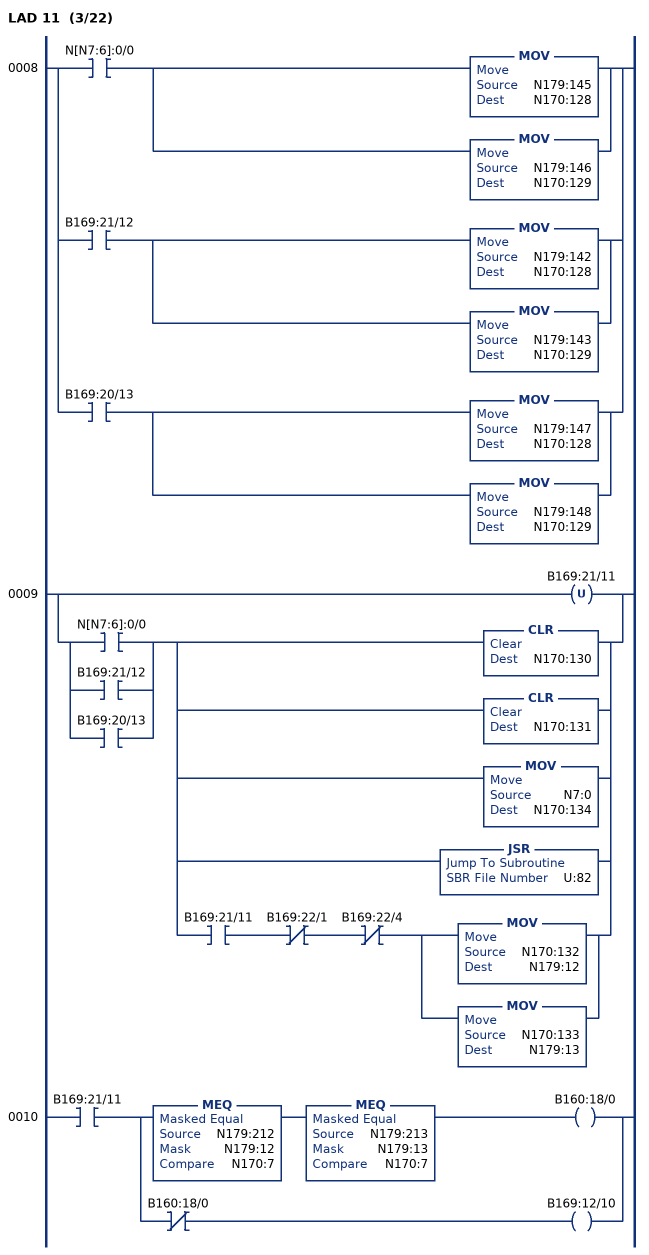
% Rung: 8 %
SOR BST XIC N[N7:6]:0/0 BST MOV N179:145 N170:128 NXB MOV N179:146 N170:129 BND NXB XIC B169:21/12 BST MOV N179:142 N170:128 NXB MOV N179:143 N170:129 BND NXB XIC B169:20/13 BST MOV N179:147 N170:128 NXB MOV N179:148 N170:129 BND BND EOR
% Rung: 9 %
SOR BST OTU B169:21/11 NXB BST XIC N[N7:6]:0/0 NXB XIC B169:21/12 NXB XIC B169:20/13 BND BST CLR N170:130 NXB CLR N170:131 NXB MOV N7:0 N170:134 NXB JSR U:82 NXB XIC B169:21/11 XIO B169:22/1 XIO B169:22/4 BST MOV N170:132 N179:12 NXB MOV N170:133 N179:13 BND BND BND EOR
% Rung: 10 %
SOR XIC B169:21/11 BST MEQ N179:212 N179:12 N170:7 MEQ N179:213 N179:13 N170:7 OTE B160:18/0 NXB XIO B160:18/0 OTE B169:12/10 BND EOR

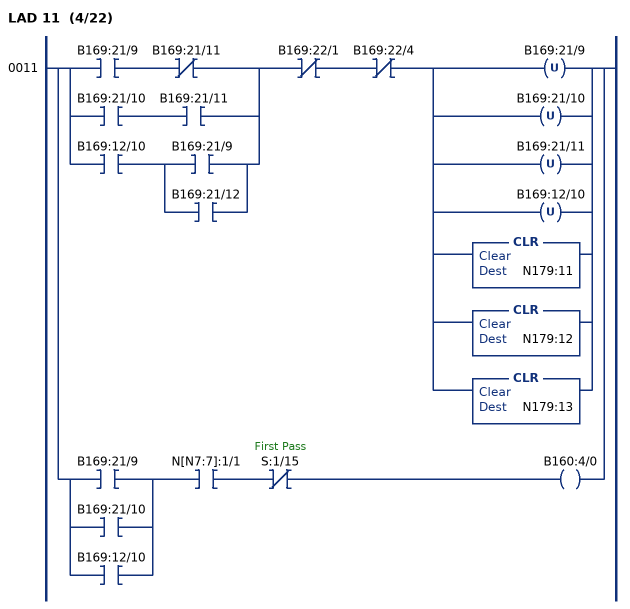
% Rung: 11 %
SOR BST BST XIC B169:21/9 XIO B169:21/11 NXB XIC B169:21/10 XIC B169:21/11 NXB XIC B169:12/10 BST XIC B169:21/9 NXB XIC B169:21/12 BND BND XIO B169:22/1 XIO B169:22/4 BST OTU B169:21/9 NXB OTU B169:21/10 NXB OTU B169:21/11 NXB OTU B169:12/10 NXB CLR N179:11 NXB CLR N179:12 NXB CLR N179:13 BND NXB BST XIC B169:21/9 NXB XIC B169:21/10 NXB XIC B169:12/10 BND XIC N[N7:7]:1/1 XIO S:1/15 OTE B160:4/0 BND EOR
%   S:1/15  "First Pass" %

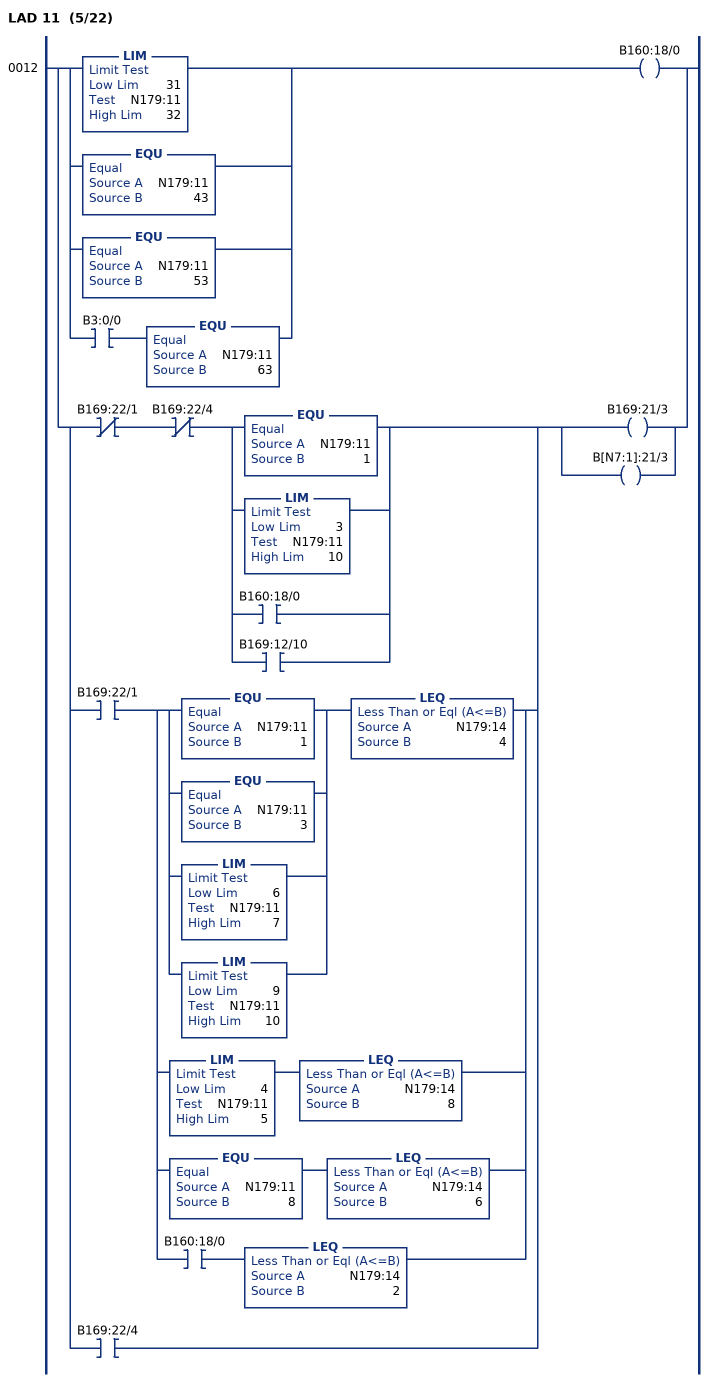
% Rung: 12 %
SOR BST BST LIM 31 N179:11 32 NXB EQU N179:11 43 NXB EQU N179:11 53 NXB XIC B3:0/0 EQU N179:11 63 BND OTE B160:18/0 NXB BST XIO B169:22/1 XIO B169:22/4 BST EQU N179:11 1 NXB LIM 3 N179:11 10 NXB XIC B160:18/0 NXB XIC B169:12/10 BND NXB XIC B169:22/1 BST BST EQU N179:11 1 NXB EQU N179:11 3 NXB LIM 6 N179:11 7 NXB LIM 9 N179:11 10 BND LEQ N179:14 4 NXB LIM 4 N179:11 5 LEQ N179:14 8 NXB EQU N179:11 8 LEQ N179:14 6 NXB XIC B160:18/0 LEQ N179:14 2 BND NXB XIC B169:22/4 BND BST OTE B169:21/3 NXB OTE B[N7:1]:21/3 BND BND EOR

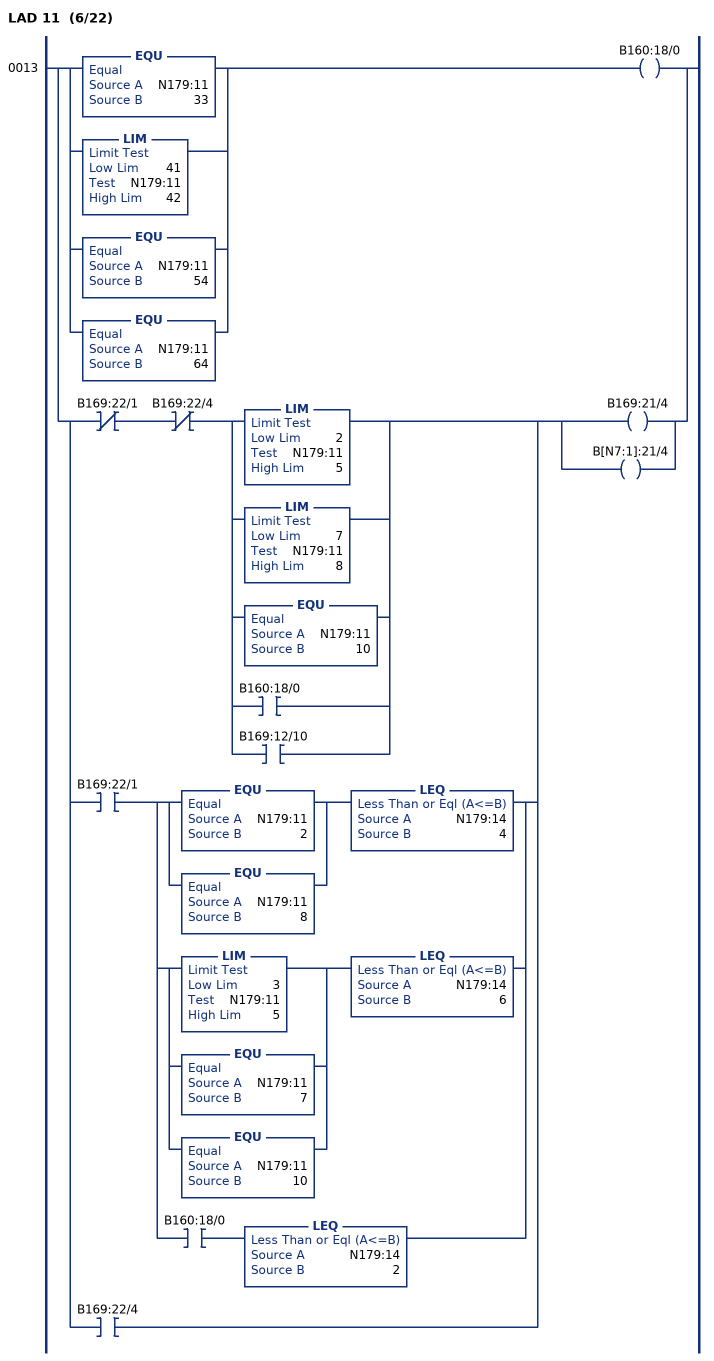
% Rung: 13 %
SOR BST BST EQU N179:11 33 NXB LIM 41 N179:11 42 NXB EQU N179:11 54 NXB EQU N179:11 64 BND OTE B160:18/0 NXB BST XIO B169:22/1 XIO B169:22/4 BST LIM 2 N179:11 5 NXB LIM 7 N179:11 8 NXB EQU N179:11 10 NXB XIC B160:18/0 NXB XIC B169:12/10 BND NXB XIC B169:22/1 BST BST EQU N179:11 2 NXB EQU N179:11 8 BND LEQ N179:14 4 NXB BST LIM 3 N179:11 5 NXB EQU N179:11 7 NXB EQU N179:11 10 BND LEQ N179:14 6 NXB XIC B160:18/0 LEQ N179:14 2 BND NXB XIC B169:22/4 BND BST OTE B169:21/4 NXB OTE B[N7:1]:21/4 BND BND EOR

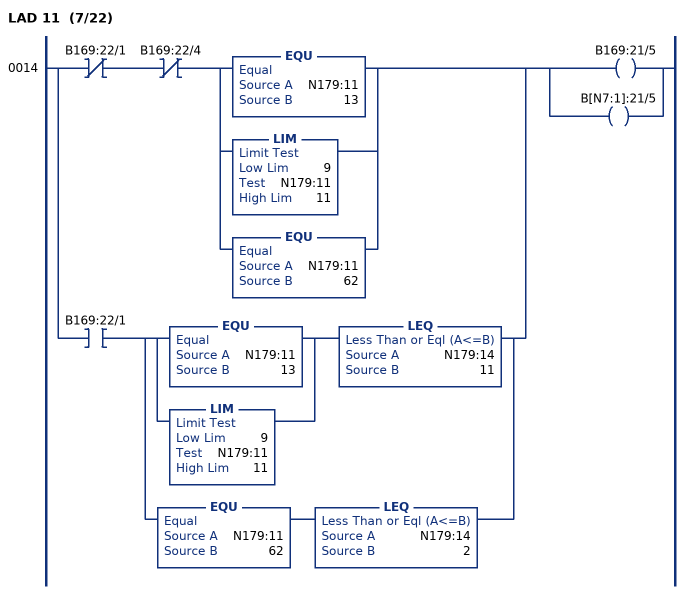
% Rung: 14 %
SOR BST XIO B169:22/1 XIO B169:22/4 BST EQU N179:11 13 NXB LIM 9 N179:11 11 NXB EQU N179:11 62 BND NXB XIC B169:22/1 BST BST EQU N179:11 13 NXB LIM 9 N179:11 11 BND LEQ N179:14 11 NXB EQU N179:11 62 LEQ N179:14 2 BND BND BST OTE B169:21/5 NXB OTE B[N7:1]:21/5 BND EOR

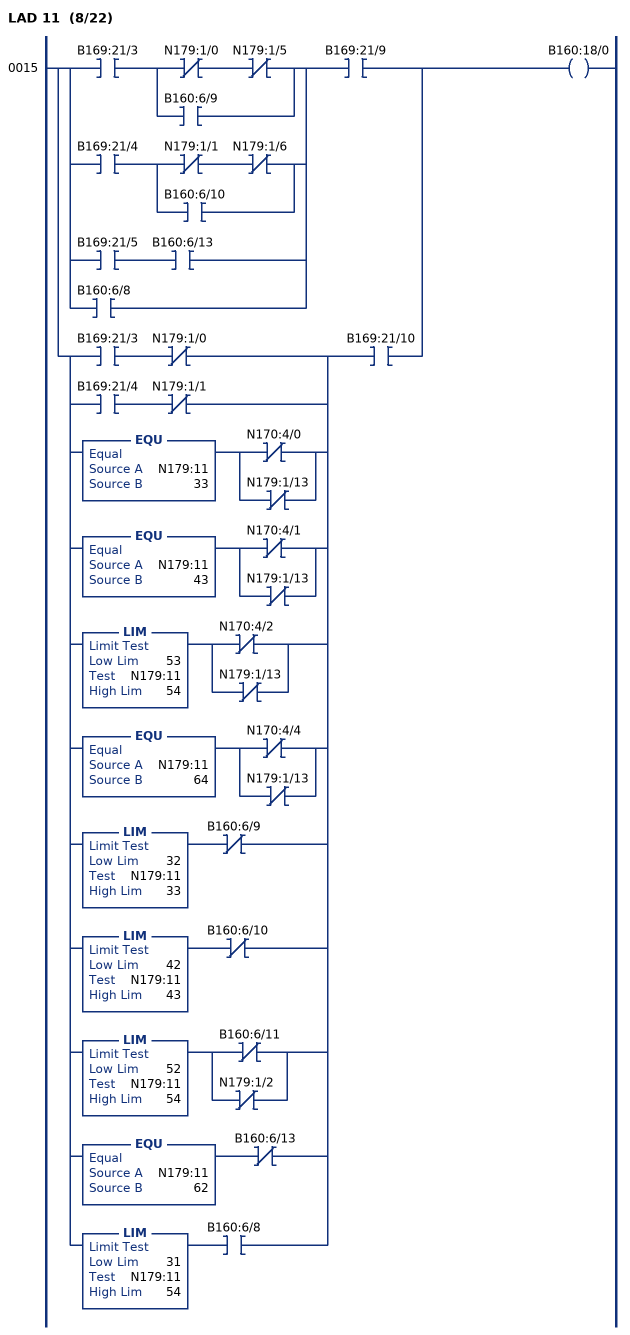
% Rung: 15 %
SOR BST BST XIC B169:21/3 BST XIO N179:1/0 XIO N179:1/5 NXB XIC B160:6/9 BND NXB XIC B169:21/4 BST XIO N179:1/1 XIO N179:1/6 NXB XIC B160:6/10 BND NXB XIC B169:21/5 XIC B160:6/13 NXB XIC B160:6/8 BND XIC B169:21/9 NXB BST XIC B169:21/3 XIO N179:1/0 NXB XIC B169:21/4 XIO N179:1/1 NXB EQU N179:11 33 BST XIO N170:4/0 NXB XIO N179:1/13 BND NXB EQU N179:11 43 BST XIO N170:4/1 NXB XIO N179:1/13 BND NXB LIM 53 N179:11 54 BST XIO N170:4/2 NXB XIO N179:1/13 BND NXB EQU N179:11 64 BST XIO N170:4/4 NXB XIO N179:1/13 BND NXB LIM 32 N179:11 33 XIO B160:6/9 NXB LIM 42 N179:11 43 XIO B160:6/10 NXB LIM 52 N179:11 54 BST XIO B160:6/11 NXB XIO N179:1/2 BND NXB EQU N179:11 62 XIO B160:6/13 NXB LIM 31 N179:11 54 XIC B160:6/8 BND XIC B169:21/10 BND OTE B160:18/0 EOR

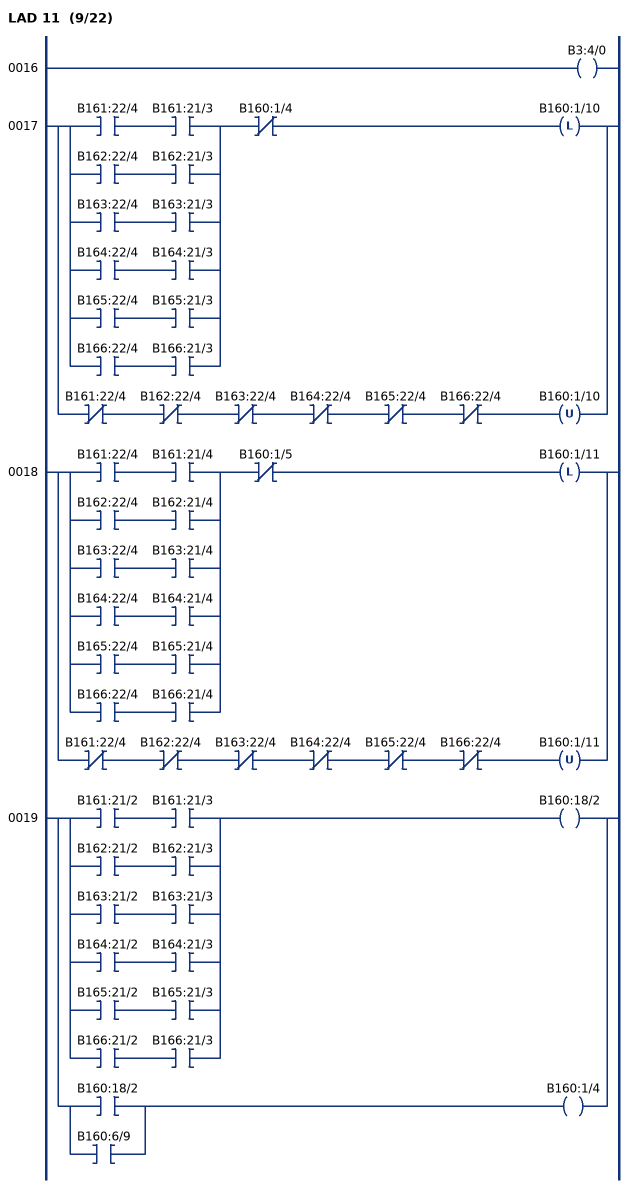
% Rung: 16 %
SOR OTE B3:4/0 EOR
% Rung: 17 %
SOR BST BST XIC B161:22/4 XIC B161:21/3 NXB XIC B162:22/4 XIC B162:21/3 NXB XIC B163:22/4 XIC B163:21/3 NXB XIC B164:22/4 XIC B164:21/3 NXB XIC B165:22/4 XIC B165:21/3 NXB XIC B166:22/4 XIC B166:21/3 BND XIO B160:1/4 OTL B160:1/10 NXB XIO B161:22/4 XIO B162:22/4 XIO B163:22/4 XIO B164:22/4 XIO B165:22/4 XIO B166:22/4 OTU B160:1/10 BND EOR
% Rung: 18 %
SOR BST BST XIC B161:22/4 XIC B161:21/4 NXB XIC B162:22/4 XIC B162:21/4 NXB XIC B163:22/4 XIC B163:21/4 NXB XIC B164:22/4 XIC B164:21/4 NXB XIC B165:22/4 XIC B165:21/4 NXB XIC B166:22/4 XIC B166:21/4 BND XIO B160:1/5 OTL B160:1/11 NXB XIO B161:22/4 XIO B162:22/4 XIO B163:22/4 XIO B164:22/4 XIO B165:22/4 XIO B166:22/4 OTU B160:1/11 BND EOR
% Rung: 19 %
SOR BST BST XIC B161:21/2 XIC B161:21/3 NXB XIC B162:21/2 XIC B162:21/3 NXB XIC B163:21/2 XIC B163:21/3 NXB XIC B164:21/2 XIC B164:21/3 NXB XIC B165:21/2 XIC B165:21/3 NXB XIC B166:21/2 XIC B166:21/3 BND OTE B160:18/2 NXB BST XIC B160:18/2 NXB XIC B160:6/9 BND OTE B160:1/4 BND EOR

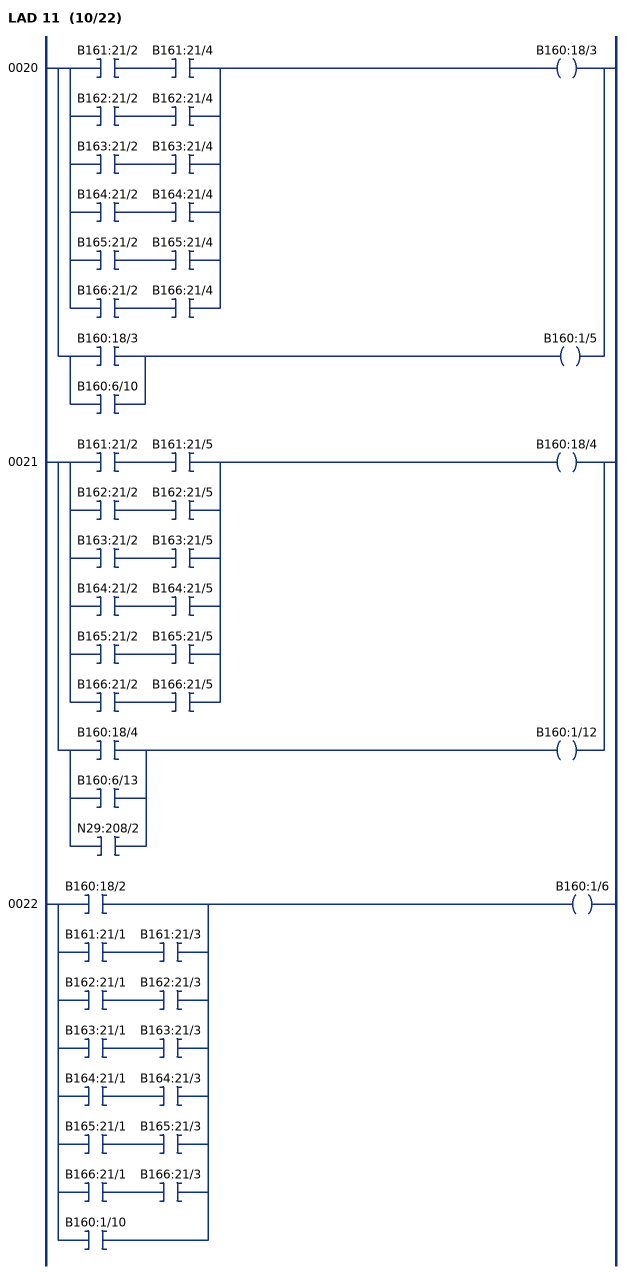
% Rung: 20 %
SOR BST BST XIC B161:21/2 XIC B161:21/4 NXB XIC B162:21/2 XIC B162:21/4 NXB XIC B163:21/2 XIC B163:21/4 NXB XIC B164:21/2 XIC B164:21/4 NXB XIC B165:21/2 XIC B165:21/4 NXB XIC B166:21/2 XIC B166:21/4 BND OTE B160:18/3 NXB BST XIC B160:18/3 NXB XIC B160:6/10 BND OTE B160:1/5 BND EOR
% Rung: 21 %
SOR BST BST XIC B161:21/2 XIC B161:21/5 NXB XIC B162:21/2 XIC B162:21/5 NXB XIC B163:21/2 XIC B163:21/5 NXB XIC B164:21/2 XIC B164:21/5 NXB XIC B165:21/2 XIC B165:21/5 NXB XIC B166:21/2 XIC B166:21/5 BND OTE B160:18/4 NXB BST XIC B160:18/4 NXB XIC B160:6/13 NXB XIC N29:208/2 BND OTE B160:1/12 BND EOR
% Rung: 22 %
SOR BST XIC B160:18/2 NXB XIC B161:21/1 XIC B161:21/3 NXB XIC B162:21/1 XIC B162:21/3 NXB XIC B163:21/1 XIC B163:21/3 NXB XIC B164:21/1 XIC B164:21/3 NXB XIC B165:21/1 XIC B165:21/3 NXB XIC B166:21/1 XIC B166:21/3 NXB XIC B160:1/10 BND OTE B160:1/6 EOR

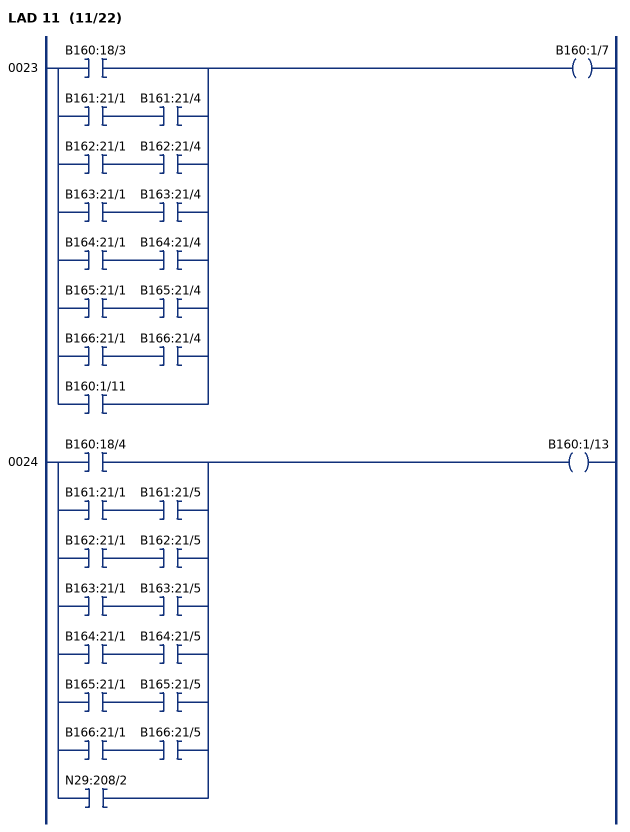
% Rung: 23 %
SOR BST XIC B160:18/3 NXB XIC B161:21/1 XIC B161:21/4 NXB XIC B162:21/1 XIC B162:21/4 NXB XIC B163:21/1 XIC B163:21/4 NXB XIC B164:21/1 XIC B164:21/4 NXB XIC B165:21/1 XIC B165:21/4 NXB XIC B166:21/1 XIC B166:21/4 NXB XIC B160:1/11 BND OTE B160:1/7 EOR
% Rung: 24 %
SOR BST XIC B160:18/4 NXB XIC B161:21/1 XIC B161:21/5 NXB XIC B162:21/1 XIC B162:21/5 NXB XIC B163:21/1 XIC B163:21/5 NXB XIC B164:21/1 XIC B164:21/5 NXB XIC B165:21/1 XIC B165:21/5 NXB XIC B166:21/1 XIC B166:21/5 NXB XIC N29:208/2 BND OTE B160:1/13 EOR

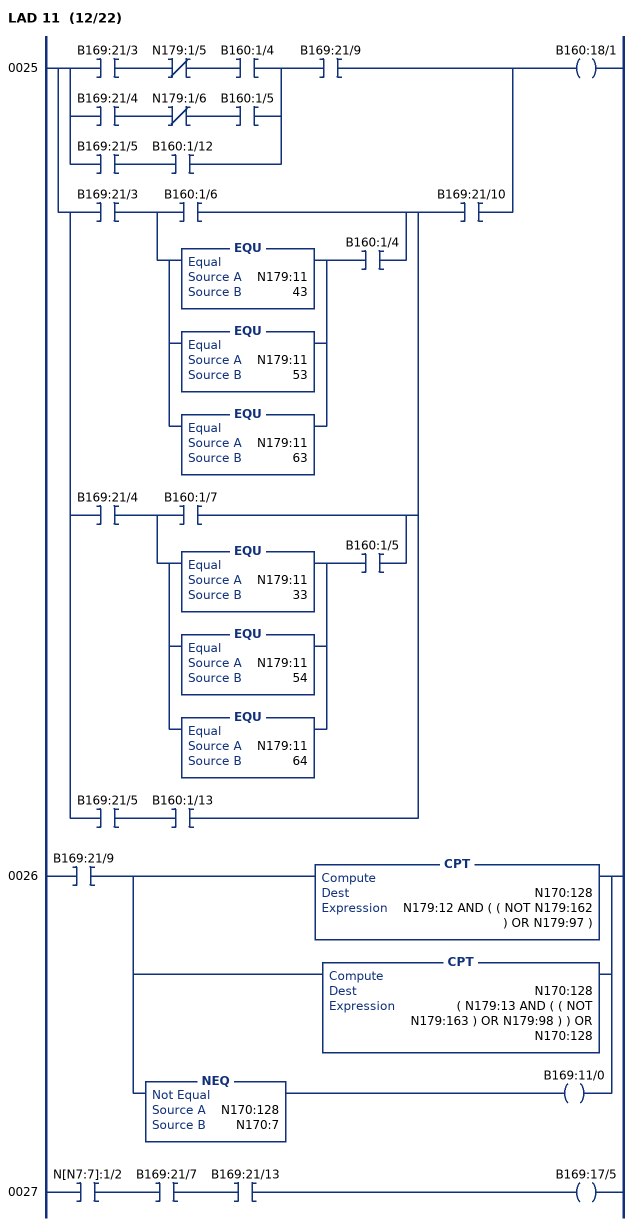
% Rung: 25 %
SOR BST BST XIC B169:21/3 XIO N179:1/5 XIC B160:1/4 NXB XIC B169:21/4 XIO N179:1/6 XIC B160:1/5 NXB XIC B169:21/5 XIC B160:1/12 BND XIC B169:21/9 NXB BST XIC B169:21/3 BST XIC B160:1/6 NXB BST EQU N179:11 43 NXB EQU N179:11 53 NXB EQU N179:11 63 BND XIC B160:1/4 BND NXB XIC B169:21/4 BST XIC B160:1/7 NXB BST EQU N179:11 33 NXB EQU N179:11 54 NXB EQU N179:11 64 BND XIC B160:1/5 BND NXB XIC B169:21/5 XIC B160:1/13 BND XIC B169:21/10 BND OTE B160:18/1 EOR
% Rung: 26 %
SOR XIC B169:21/9 BST CPT N170:128 " N179:12 AND ( ( NOT N179:162 ) OR N179:97 ) " NXB CPT N170:128 " ( N179:13 AND ( ( NOT N179:163 ) OR N179:98 ) ) OR N170:128 " NXB NEQ N170:128 N170:7 OTE B169:11/0 BND EOR
% Rung: 27 %
SOR XIC N[N7:7]:1/2 XIC B169:21/7 XIC B169:21/13 OTE B169:17/5 EOR

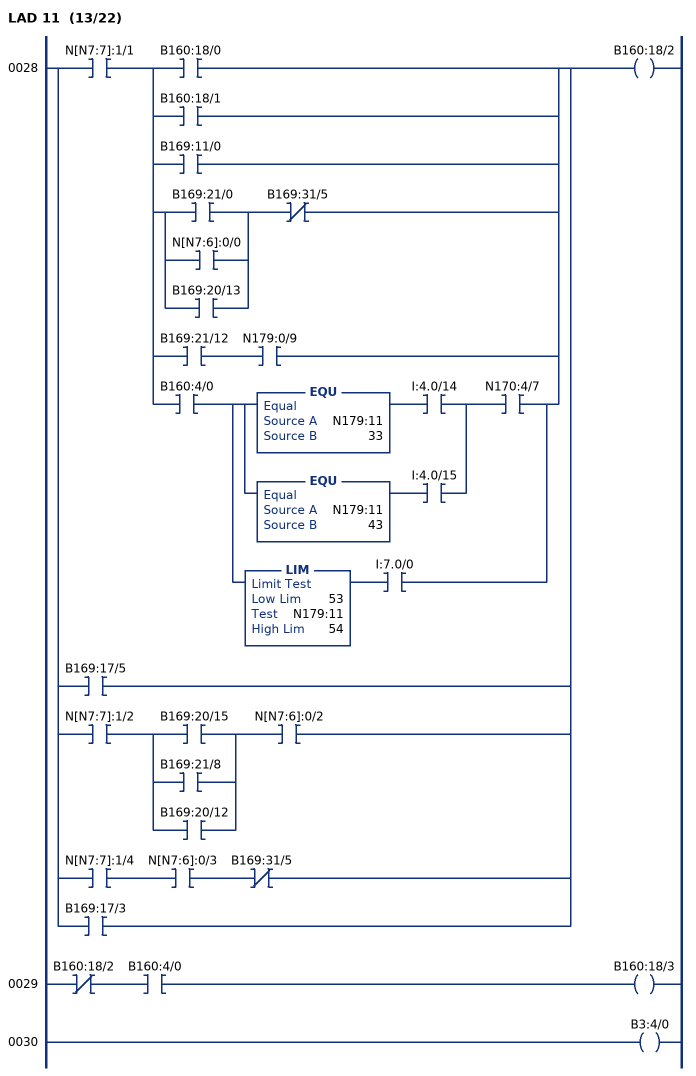
% Rung: 28 %
SOR BST XIC N[N7:7]:1/1 BST XIC B160:18/0 NXB XIC B160:18/1 NXB XIC B169:11/0 NXB BST XIC B169:21/0 NXB XIC N[N7:6]:0/0 NXB XIC B169:20/13 BND XIO B169:31/5 NXB XIC B169:21/12 XIC N179:0/9 NXB XIC B160:4/0 BST BST EQU N179:11 33 XIC I:4.0/14 NXB EQU N179:11 43 XIC I:4.0/15 BND XIC N170:4/7 NXB LIM 53 N179:11 54 XIC I:7.0/0 BND BND NXB BST XIC B169:17/5 NXB XIC N[N7:7]:1/2 BST XIC B169:20/15 NXB XIC B169:21/8 NXB XIC B169:20/12 BND XIC N[N7:6]:0/2 BND NXB XIC N[N7:7]:1/4 XIC N[N7:6]:0/3 XIO B169:31/5 NXB XIC B169:17/3 BND OTE B160:18/2 EOR
% Rung: 29 %
SOR XIO B160:18/2 XIC B160:4/0 OTE B160:18/3 EOR
% Rung: 30 %
SOR OTE B3:4/0 EOR

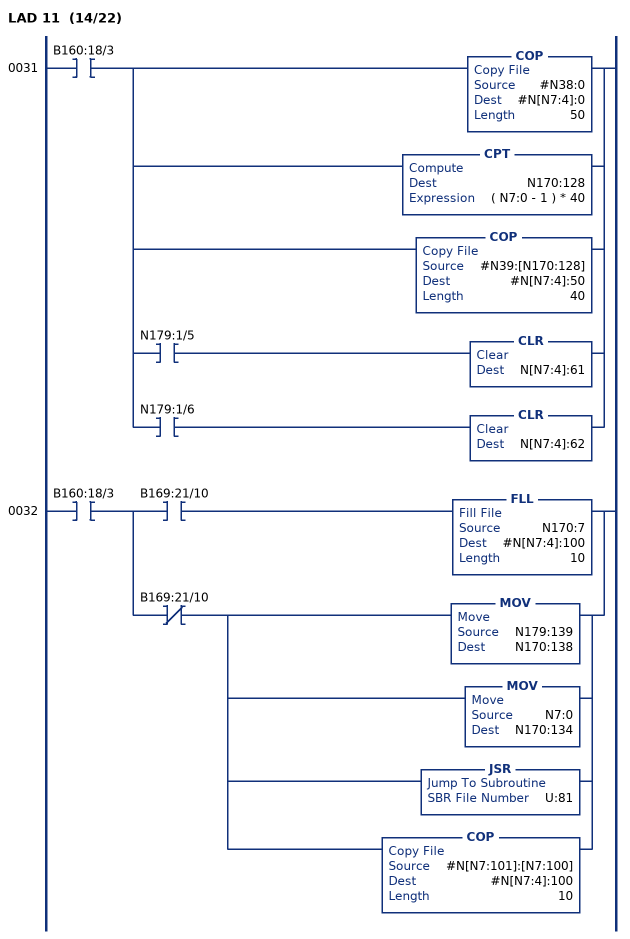
% Rung: 31 %
SOR XIC B160:18/3 BST COP #N38:0 #N[N7:4]:0 50 NXB CPT N170:128 " ( N7:0 - 1 ) * 40 " NXB COP #N39:[N170:128] #N[N7:4]:50 40 NXB XIC N179:1/5 CLR N[N7:4]:61 NXB XIC N179:1/6 CLR N[N7:4]:62 BND EOR
% Rung: 32 %
SOR XIC B160:18/3 BST XIC B169:21/10 FLL N170:7 #N[N7:4]:100 10 NXB XIO B169:21/10 BST MOV N179:139 N170:138 NXB MOV N7:0 N170:134 NXB JSR U:81 NXB COP #N[N7:101]:[N7:100] #N[N7:4]:100 10 BND BND EOR

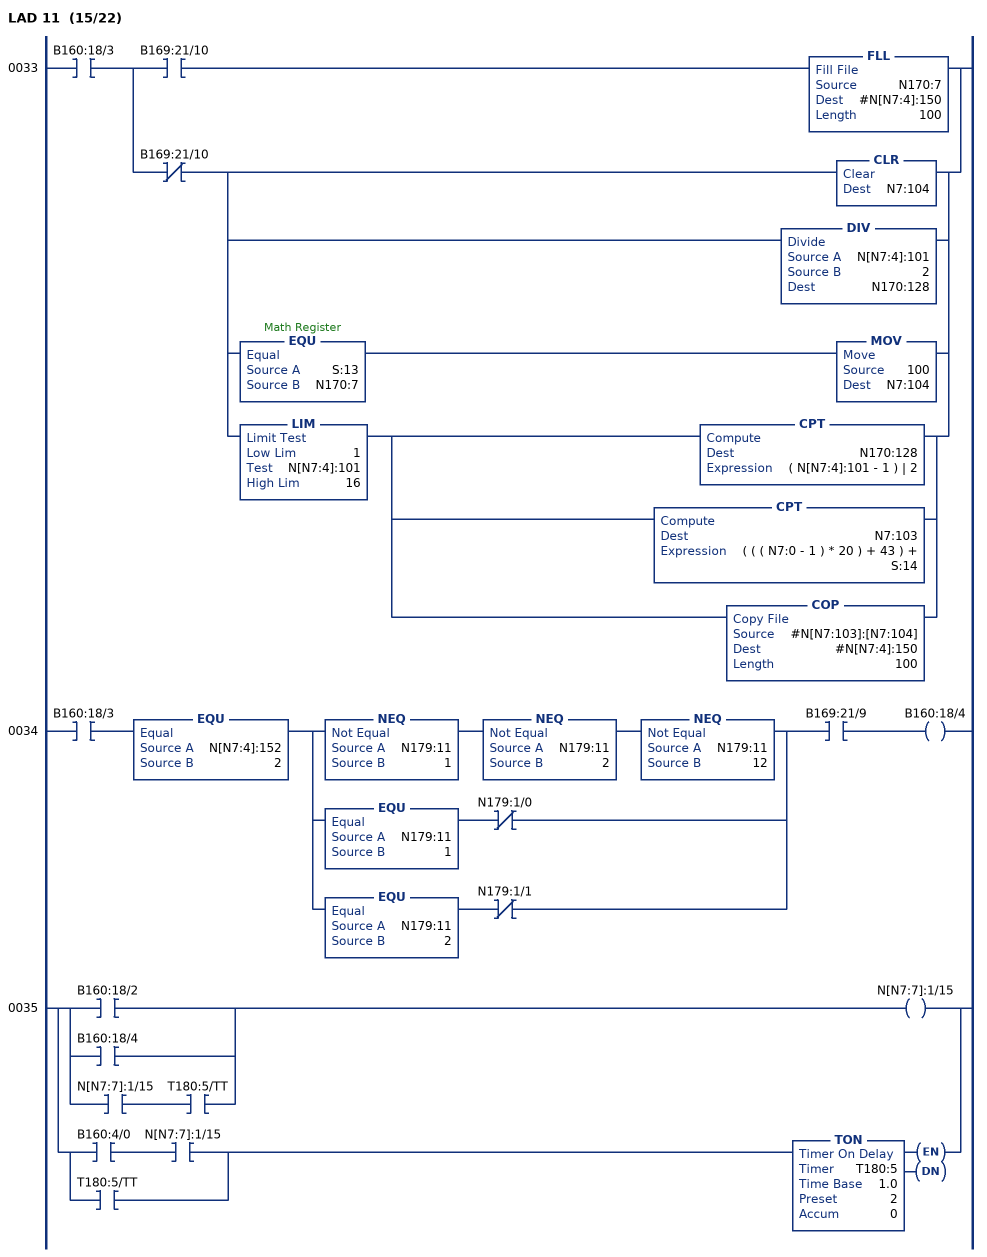
% Rung: 33 %
SOR XIC B160:18/3 BST XIC B169:21/10 FLL N170:7 #N[N7:4]:150 100 NXB XIO B169:21/10 BST CLR N7:104 NXB DIV N[N7:4]:101 2 N170:128 NXB EQU S:13 N170:7 MOV 100 N7:104 NXB LIM 1 N[N7:4]:101 16 BST CPT N170:128 " ( N[N7:4]:101 - 1 ) | 2 " NXB CPT N7:103 " ( ( ( N7:0 - 1 ) * 20 ) + 43 ) + S:14 " NXB COP #N[N7:103]:[N7:104] #N[N7:4]:150 100 BND BND BND EOR
%   S:13  "Math Register" %
%   S:14  "Math Register" %
% Rung: 34 %
SOR XIC B160:18/3 EQU N[N7:4]:152 2 BST NEQ N179:11 1 NEQ N179:11 2 NEQ N179:11 12 NXB EQU N179:11 1 XIO N179:1/0 NXB EQU N179:11 2 XIO N179:1/1 BND XIC B169:21/9 OTE B160:18/4 EOR
% Rung: 35 %
SOR BST BST XIC B160:18/2 NXB XIC B160:18/4 NXB XIC N[N7:7]:1/15 XIC T180:5/TT BND OTE N[N7:7]:1/15 NXB BST XIC B160:4/0 XIC N[N7:7]:1/15 NXB XIC T180:5/TT BND TON T180:5 1.0 2 0 BND EOR

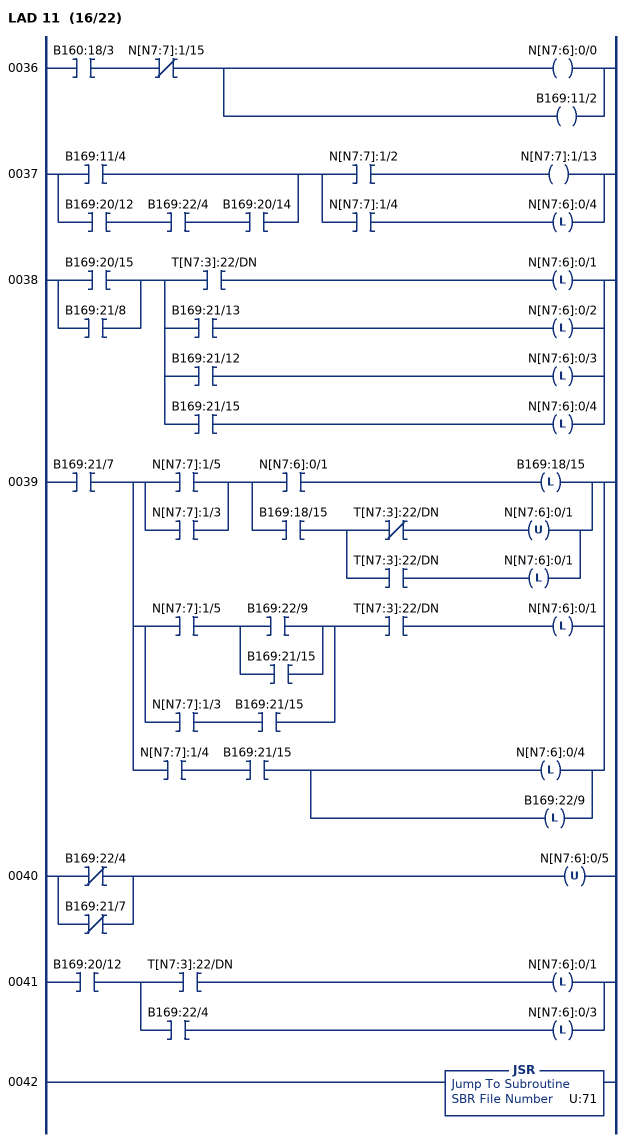
% Rung: 36 %
SOR XIC B160:18/3 XIO N[N7:7]:1/15 BST OTE N[N7:6]:0/0 NXB OTE B169:11/2 BND EOR
% Rung: 37 %
SOR BST XIC B169:11/4 NXB XIC B169:20/12 XIC B169:22/4 XIC B169:20/14 BND BST XIC N[N7:7]:1/2 OTE N[N7:7]:1/13 NXB XIC N[N7:7]:1/4 OTL N[N7:6]:0/4 BND EOR
% Rung: 38 %
SOR BST XIC B169:20/15 NXB XIC B169:21/8 BND BST XIC T[N7:3]:22/DN OTL N[N7:6]:0/1 NXB XIC B169:21/13 OTL N[N7:6]:0/2 NXB XIC B169:21/12 OTL N[N7:6]:0/3 NXB XIC B169:21/15 OTL N[N7:6]:0/4 BND EOR
% Rung: 39 %
SOR XIC B169:21/7 BST BST XIC N[N7:7]:1/5 NXB XIC N[N7:7]:1/3 BND BST XIC N[N7:6]:0/1 OTL B169:18/15 NXB XIC B169:18/15 BST XIO T[N7:3]:22/DN OTU N[N7:6]:0/1 NXB XIC T[N7:3]:22/DN OTL N[N7:6]:0/1 BND BND NXB BST XIC N[N7:7]:1/5 BST XIC B169:22/9 NXB XIC B169:21/15 BND NXB XIC N[N7:7]:1/3 XIC B169:21/15 BND XIC T[N7:3]:22/DN OTL N[N7:6]:0/1 NXB XIC N[N7:7]:1/4 XIC B169:21/15 BST OTL N[N7:6]:0/4 NXB OTL B169:22/9 BND BND EOR
% Rung: 40 %
SOR BST XIO B169:22/4 NXB XIO B169:21/7 BND OTU N[N7:6]:0/5 EOR
% Rung: 41 %
SOR XIC B169:20/12 BST XIC T[N7:3]:22/DN OTL N[N7:6]:0/1 NXB XIC B169:22/4 OTL N[N7:6]:0/3 BND EOR
% Rung: 42 %
SOR JSR U:71 EOR

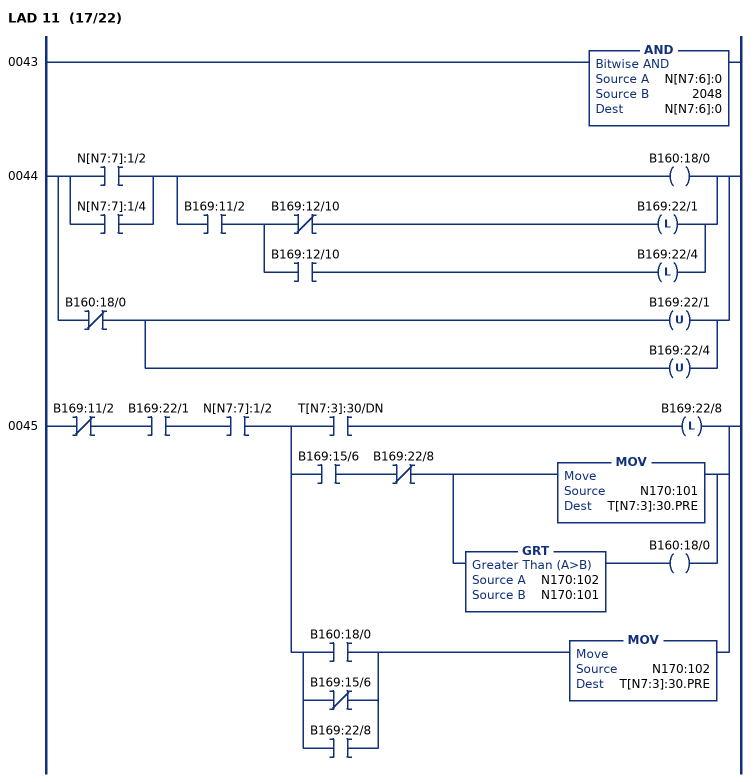
% Rung: 43 %
SOR AND N[N7:6]:0 2048 N[N7:6]:0 EOR
% Rung: 44 %
SOR BST BST XIC N[N7:7]:1/2 NXB XIC N[N7:7]:1/4 BND BST OTE B160:18/0 NXB XIC B169:11/2 BST XIO B169:12/10 OTL B169:22/1 NXB XIC B169:12/10 OTL B169:22/4 BND BND NXB XIO B160:18/0 BST OTU B169:22/1 NXB OTU B169:22/4 BND BND EOR
% Rung: 45 %
SOR XIO B169:11/2 XIC B169:22/1 XIC N[N7:7]:1/2 BST XIC T[N7:3]:30/DN OTL B169:22/8 NXB XIC B169:15/6 XIO B169:22/8 BST MOV N170:101 T[N7:3]:30.PRE NXB GRT N170:102 N170:101 OTE B160:18/0 BND NXB BST XIC B160:18/0 NXB XIO B169:15/6 NXB XIC B169:22/8 BND MOV N170:102 T[N7:3]:30.PRE BND EOR

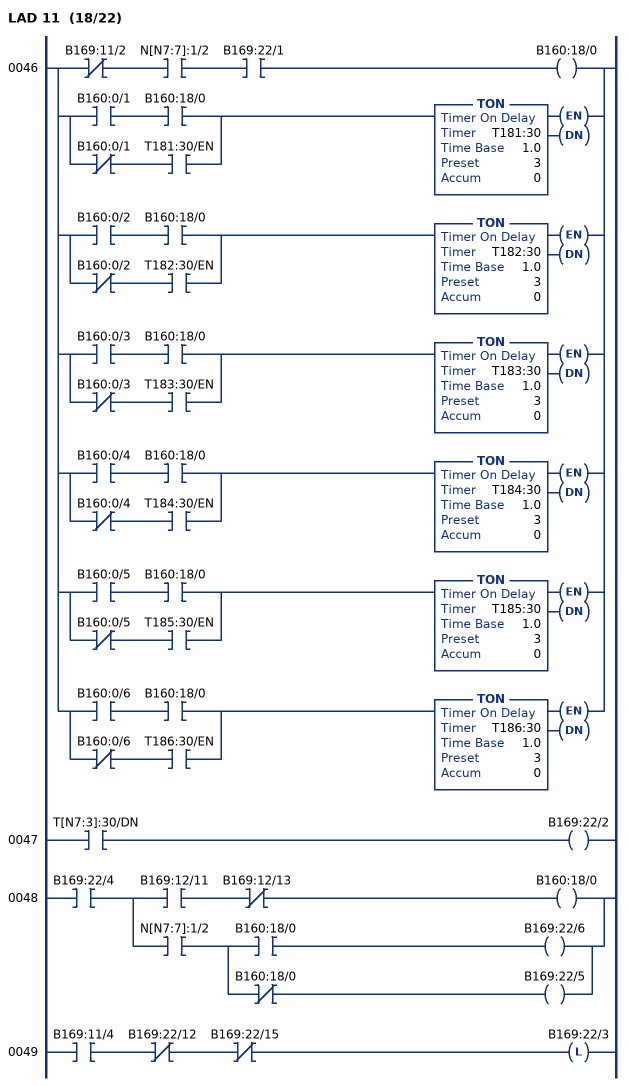
% Rung: 46 %
SOR BST XIO B169:11/2 XIC N[N7:7]:1/2 XIC B169:22/1 OTE B160:18/0 NXB BST XIC B160:0/1 XIC B160:18/0 NXB XIO B160:0/1 XIC T181:30/EN BND TON T181:30 1.0 3 0 NXB BST XIC B160:0/2 XIC B160:18/0 NXB XIO B160:0/2 XIC T182:30/EN BND TON T182:30 1.0 3 0 NXB BST XIC B160:0/3 XIC B160:18/0 NXB XIO B160:0/3 XIC T183:30/EN BND TON T183:30 1.0 3 0 NXB BST XIC B160:0/4 XIC B160:18/0 NXB XIO B160:0/4 XIC T184:30/EN BND TON T184:30 1.0 3 0 NXB BST XIC B160:0/5 XIC B160:18/0 NXB XIO B160:0/5 XIC T185:30/EN BND TON T185:30 1.0 3 0 NXB BST XIC B160:0/6 XIC B160:18/0 NXB XIO B160:0/6 XIC T186:30/EN BND TON T186:30 1.0 3 0 BND EOR
% Rung: 47 %
SOR XIC T[N7:3]:30/DN OTE B169:22/2 EOR
% Rung: 48 %
SOR XIC B169:22/4 BST XIC B169:12/11 XIO B169:12/13 OTE B160:18/0 NXB XIC N[N7:7]:1/2 BST XIC B160:18/0 OTE B169:22/6 NXB XIO B160:18/0 OTE B169:22/5 BND BND EOR
% Rung: 49 %
SOR XIC B169:11/4 XIO B169:22/12 XIO B169:22/15 OTL B169:22/3 EOR

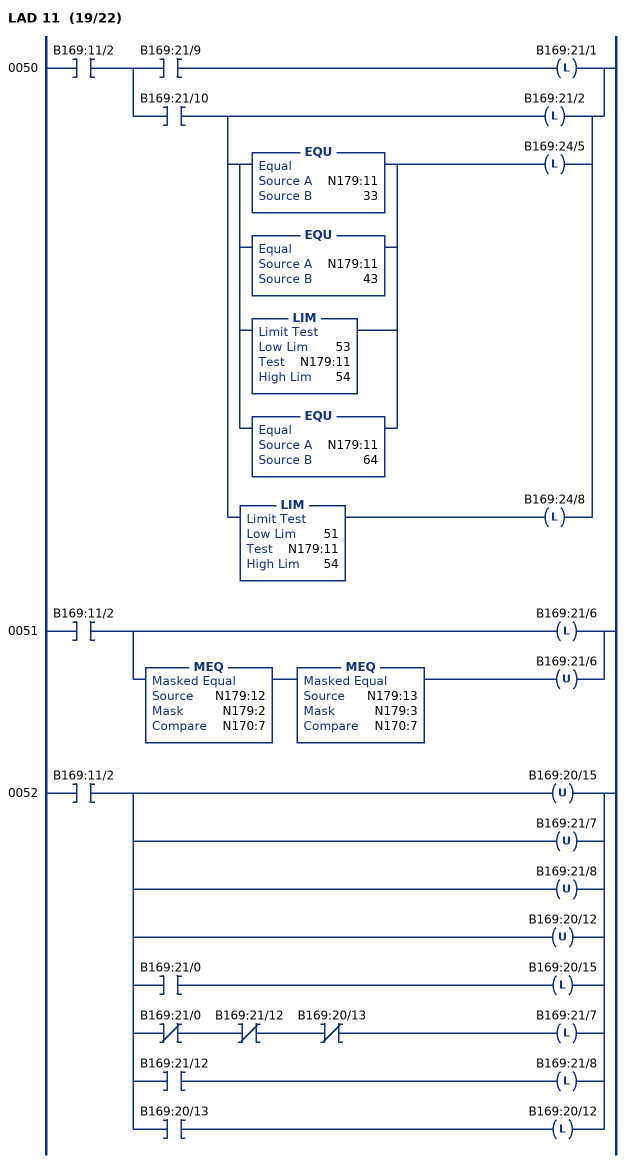
% Rung: 50 %
SOR XIC B169:11/2 BST XIC B169:21/9 OTL B169:21/1 NXB XIC B169:21/10 BST OTL B169:21/2 NXB BST EQU N179:11 33 NXB EQU N179:11 43 NXB LIM 53 N179:11 54 NXB EQU N179:11 64 BND OTL B169:24/5 NXB LIM 51 N179:11 54 OTL B169:24/8 BND BND EOR
% Rung: 51 %
SOR XIC B169:11/2 BST OTL B169:21/6 NXB MEQ N179:12 N179:2 N170:7 MEQ N179:13 N179:3 N170:7 OTU B169:21/6 BND EOR
% Rung: 52 %
SOR XIC B169:11/2 BST BST OTU B169:20/15 NXB OTU B169:21/7 NXB OTU B169:21/8 NXB OTU B169:20/12 BND NXB XIC B169:21/0 OTL B169:20/15 NXB XIO B169:21/0 XIO B169:21/12 XIO B169:20/13 OTL B169:21/7 NXB XIC B169:21/12 OTL B169:21/8 NXB XIC B169:20/13 OTL B169:20/12 BND EOR

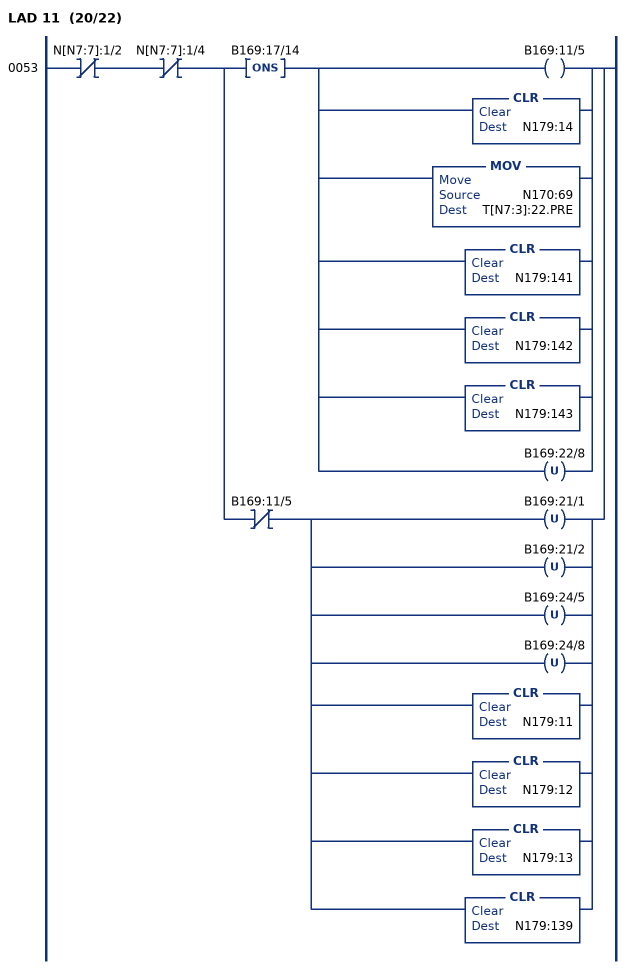
% Rung: 53 %
SOR XIO N[N7:7]:1/2 XIO N[N7:7]:1/4 BST OSR B169:17/14 BST OTE B169:11/5 NXB CLR N179:14 NXB MOV N170:69 T[N7:3]:22.PRE NXB CLR N179:141 NXB CLR N179:142 NXB CLR N179:143 NXB OTU B169:22/8 BND NXB XIO B169:11/5 BST OTU B169:21/1 NXB OTU B169:21/2 NXB OTU B169:24/5 NXB OTU B169:24/8 NXB CLR N179:11 NXB CLR N179:12 NXB CLR N179:13 NXB CLR N179:139 BND BND EOR

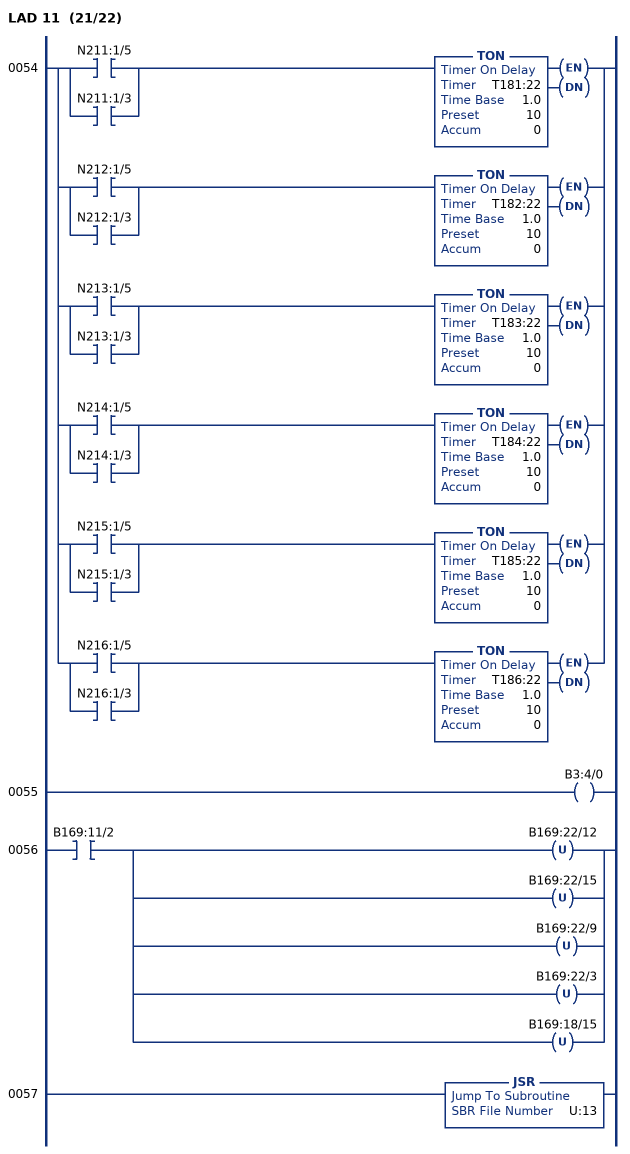
% Rung: 54 %
SOR BST BST XIC N211:1/5 NXB XIC N211:1/3 BND TON T181:22 1.0 10 0 NXB BST XIC N212:1/5 NXB XIC N212:1/3 BND TON T182:22 1.0 10 0 NXB BST XIC N213:1/5 NXB XIC N213:1/3 BND TON T183:22 1.0 10 0 NXB BST XIC N214:1/5 NXB XIC N214:1/3 BND TON T184:22 1.0 10 0 NXB BST XIC N215:1/5 NXB XIC N215:1/3 BND TON T185:22 1.0 10 0 NXB BST XIC N216:1/5 NXB XIC N216:1/3 BND TON T186:22 1.0 10 0 BND EOR
% Rung: 55 %
SOR OTE B3:4/0 EOR
% Rung: 56 %
SOR XIC B169:11/2 BST OTU B169:22/12 NXB OTU B169:22/15 NXB OTU B169:22/9 NXB OTU B169:22/3 NXB OTU B169:18/15 BND EOR
% Rung: 57 %
SOR JSR U:13 EOR

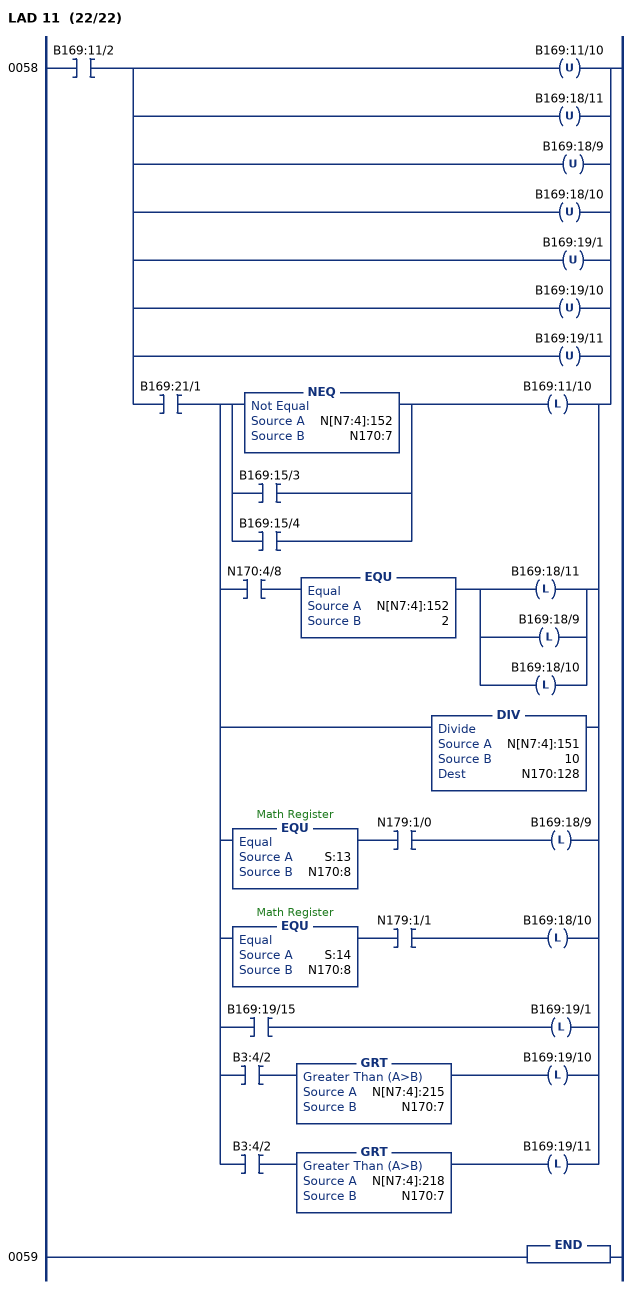
% Rung: 58 %
SOR XIC B169:11/2 BST BST OTU B169:11/10 NXB OTU B169:18/11 NXB OTU B169:18/9 NXB OTU B169:18/10 NXB OTU B169:19/1 NXB OTU B169:19/10 NXB OTU B169:19/11 BND NXB XIC B169:21/1 BST BST NEQ N[N7:4]:152 N170:7 NXB XIC B169:15/3 NXB XIC B169:15/4 BND OTL B169:11/10 NXB XIC N170:4/8 EQU N[N7:4]:152 2 BST OTL B169:18/11 NXB OTL B169:18/9 NXB OTL B169:18/10 BND NXB BST DIV N[N7:4]:151 10 N170:128 NXB EQU S:13 N170:8 XIC N179:1/0 OTL B169:18/9 NXB EQU S:14 N170:8 XIC N179:1/1 OTL B169:18/10 BND NXB XIC B169:19/15 OTL B169:19/1 NXB XIC B3:4/2 GRT N[N7:4]:215 N170:7 OTL B169:19/10 NXB XIC B3:4/2 GRT N[N7:4]:218 N170:7 OTL B169:19/11 BND BND EOR
%   S:13  "Math Register" %
%   S:14  "Math Register" %
% Rung: 59 %
SOR END EOR

LADDER 13
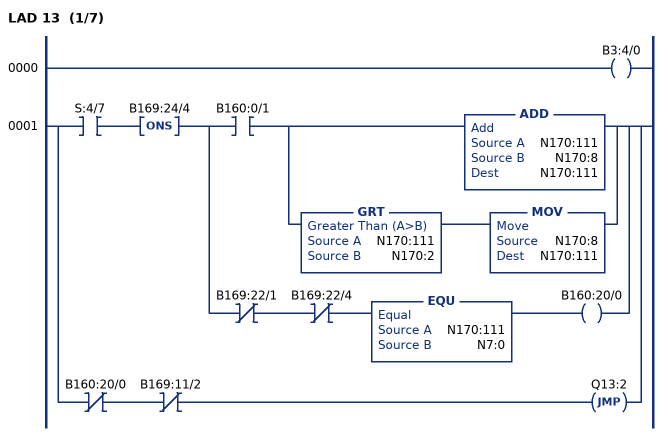
% Rung: 0 %
SOR OTE B3:4/0 EOR
% Rung: 1 %
SOR BST XIC S:4/7 OSR B169:24/4 BST XIC B160:0/1 BST ADD N170:111 N170:8 N170:111 NXB GRT N170:111 N170:2 MOV N170:8 N170:111 BND NXB XIO B169:22/1 XIO B169:22/4 EQU N170:111 N7:0 OTE B160:20/0 BND NXB XIO B160:20/0 XIO B169:11/2 JMP Q13:2 BND EOR

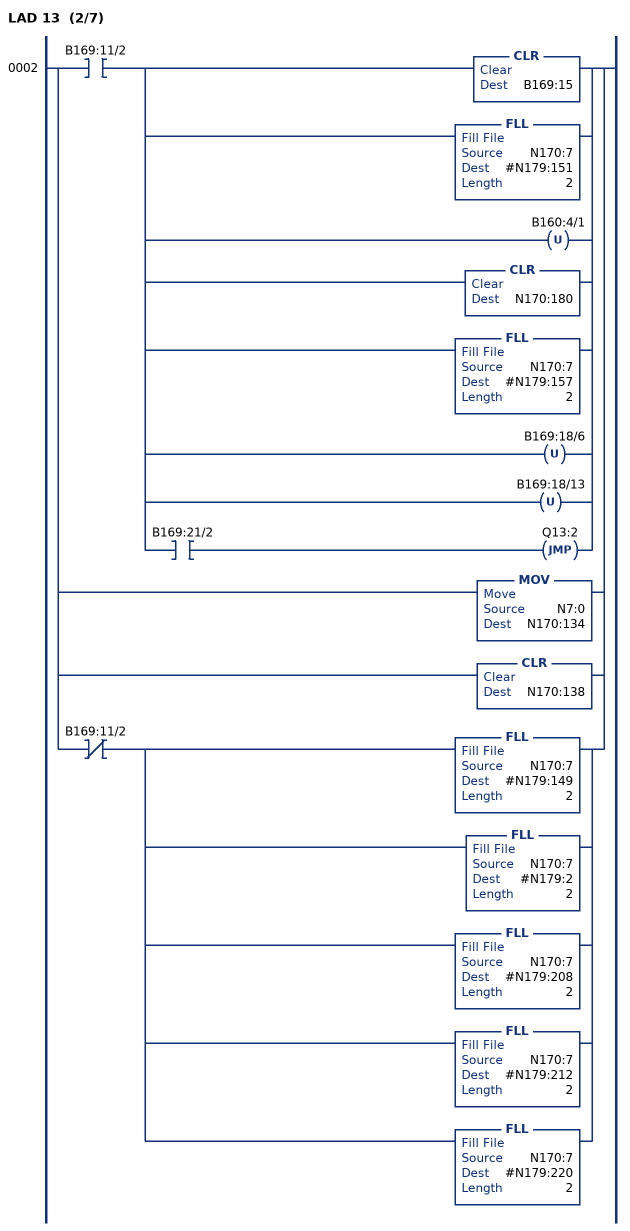
% Rung: 2 %
SOR BST XIC B169:11/2 BST BST CLR B169:15 NXB FLL N170:7 #N179:151 2 NXB OTU B160:4/1 NXB CLR N170:180 NXB FLL N170:7 #N179:157 2 NXB OTU B169:18/6 NXB OTU B169:18/13 BND NXB XIC B169:21/2 JMP Q13:2 BND NXB MOV N7:0 N170:134 NXB CLR N170:138 NXB XIO B169:11/2 BST FLL N170:7 #N179:149 2 NXB FLL N170:7 #N179:2 2 NXB FLL N170:7 #N179:208 2 NXB FLL N170:7 #N179:212 2 NXB FLL N170:7 #N179:220 2 BND BND EOR

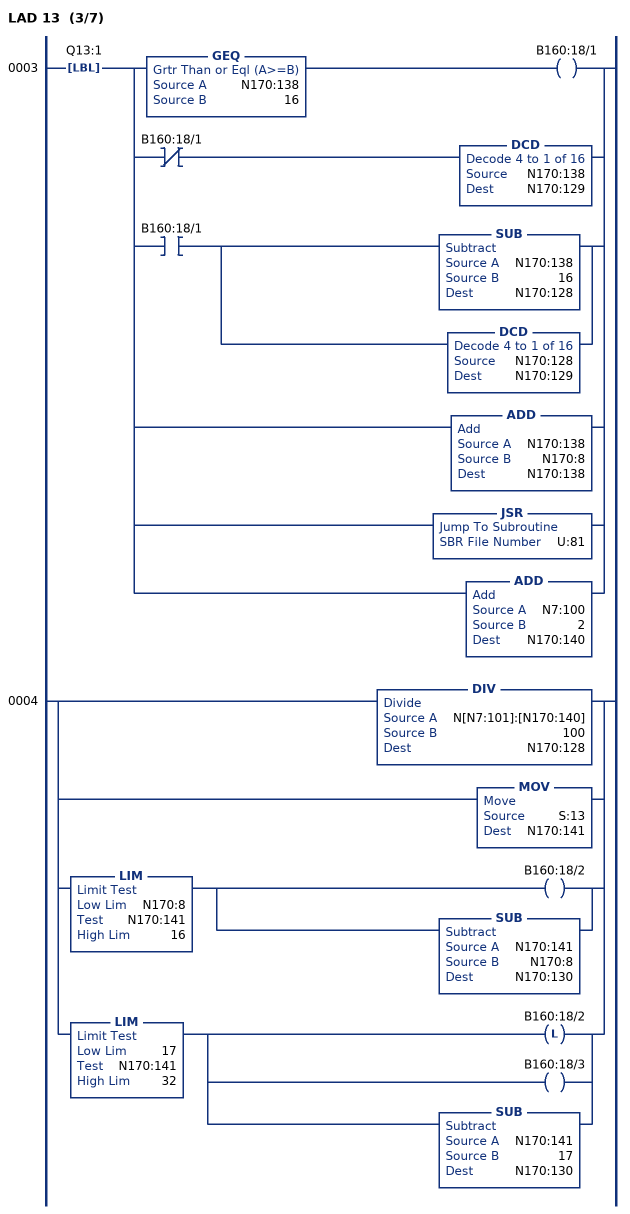
% Rung: 3 %
SOR LBL Q13:1 BST GEQ N170:138 16 OTE B160:18/1 NXB XIO B160:18/1 DCD N170:138 N170:129 NXB XIC B160:18/1 BST SUB N170:138 16 N170:128 NXB DCD N170:128 N170:129 BND NXB ADD N170:138 N170:8 N170:138 NXB JSR U:81 NXB ADD N7:100 2 N170:140 BND EOR
% Rung: 4 %
SOR BST BST DIV N[N7:101]:[N170:140] 100 N170:128 NXB MOV S:13 N170:141 BND NXB BST LIM N170:8 N170:141 16 BST OTE B160:18/2 NXB SUB N170:141 N170:8 N170:130 BND NXB LIM 17 N170:141 32 BST OTL B160:18/2 NXB OTE B160:18/3 NXB SUB N170:141 17 N170:130 BND BND BND EOR
%   S:13  "Math Register" %

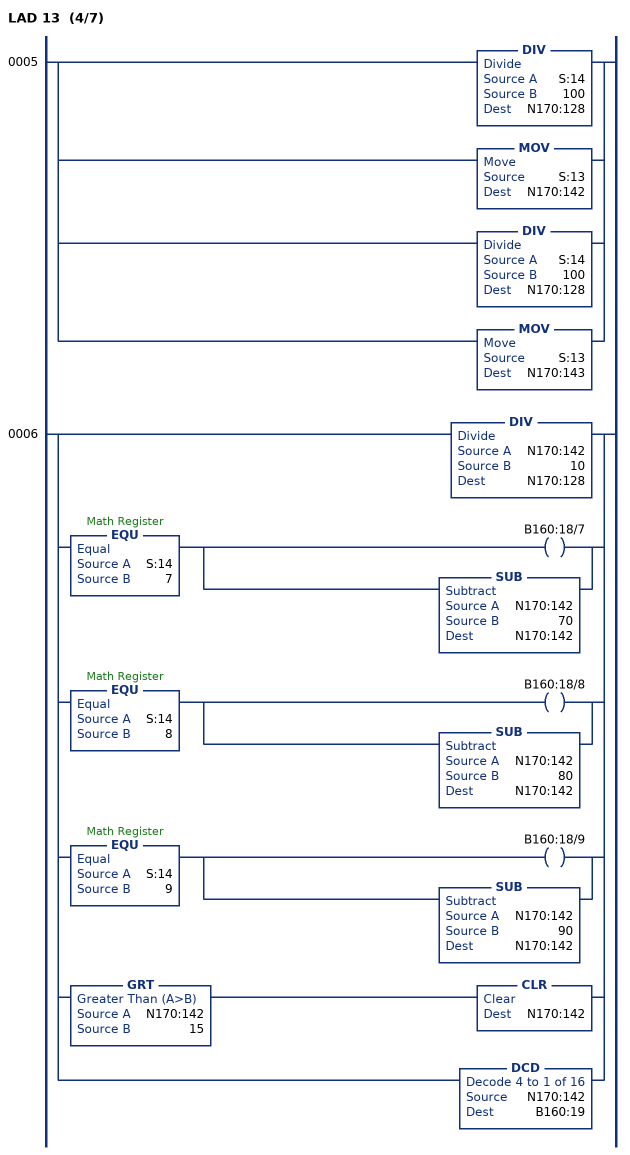
% Rung: 5 %
SOR BST BST DIV S:14 100 N170:128 NXB MOV S:13 N170:142 BND NXB BST DIV S:14 100 N170:128 NXB MOV S:13 N170:143 BND BND EOR
%   S:14  "Math Register" %
%   S:13  "Math Register" %
% Rung: 6 %
SOR BST BST DIV N170:142 10 N170:128 NXB EQU S:14 7 BST OTE B160:18/7 NXB SUB N170:142 70 N170:142 BND NXB EQU S:14 8 BST OTE B160:18/8 NXB SUB N170:142 80 N170:142 BND NXB EQU S:14 9 BST OTE B160:18/9 NXB SUB N170:142 90 N170:142 BND BND NXB BST GRT N170:142 15 CLR N170:142 NXB DCD N170:142 B160:19 BND BND EOR
%   S:14  "Math Register" %

